Staubli VAL3: getCycleTime.pgx

program getCycleTime()
begin
  //
  cls()
  //
  nCycleTime=$getCycleTime()
  //
  gotoxy(1,0)
  put("当前系统周期(s)："+toString("4.3",nCycleTime))
end
